TYPE ST_MainProcessSupervisorPar :
STRUCT
    rLevelMinSP               : REAL;
    rLevelMaxSP               : REAL;
END_STRUCT
END_TYPE

(* stored: Version 1.1.0.1, ProductVersion 3.1.4024.16
   DUT ST_MainProcessSupervisorPar: Id {17192ac8-8a54-413a-9858-b0f6eafd124a} *)
